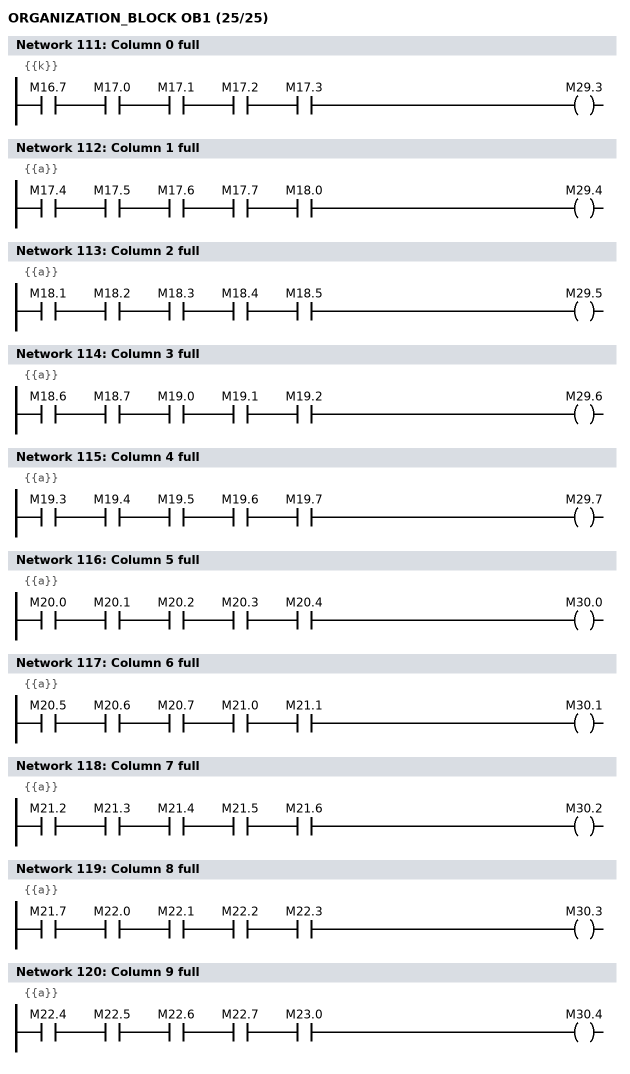

       A    M16.7
       A    M17.0
       A    M17.1
       A    M17.2
       A    M17.3
       =    M29.3
NETWORK
TITLE=Column 1 full
//{{a}}

       A    M17.4
       A    M17.5
       A    M17.6
       A    M17.7
       A    M18.0
       =    M29.4
NETWORK
TITLE=Column 2 full
//{{a}}

       A    M18.1
       A    M18.2
       A    M18.3
       A    M18.4
       A    M18.5
       =    M29.5
NETWORK
TITLE=Column 3 full
//{{a}}

       A    M18.6
       A    M18.7
       A    M19.0
       A    M19.1
       A    M19.2
       =    M29.6
NETWORK
TITLE=Column 4 full
//{{a}}

       A    M19.3
       A    M19.4
       A    M19.5
       A    M19.6
       A    M19.7
       =    M29.7
NETWORK
TITLE=Column 5 full
//{{a}}

       A    M20.0
       A    M20.1
       A    M20.2
       A    M20.3
       A    M20.4
       =    M30.0
NETWORK
TITLE=Column 6 full
//{{a}}

       A    M20.5
       A    M20.6
       A    M20.7
       A    M21.0
       A    M21.1
       =    M30.1
NETWORK
TITLE=Column 7 full
//{{a}}

       A    M21.2
       A    M21.3
       A    M21.4
       A    M21.5
       A    M21.6
       =    M30.2
NETWORK
TITLE=Column 8 full
//{{a}}

       A    M21.7
       A    M22.0
       A    M22.1
       A    M22.2
       A    M22.3
       =    M30.3
NETWORK
TITLE=Column 9 full
//{{a}}

       A    M22.4
       A    M22.5
       A    M22.6
       A    M22.7
       A    M23.0
       =    M30.4
END_ORGANIZATION_BLOCK
